(* PLC project  *)

PROGRAM P

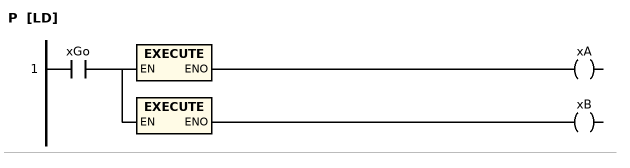
(* LD diagram, written out as Structured Text *)
IF xGo THEN
  nCount := nCount + 1;
END_IF;
xA := xGo;
IF xGo THEN
  nCount := nCount + 1;
END_IF;
xB := xGo;
END_PROGRAM
